PROGRAM MAIN
VAR
END_VAR

FillBox();
Vision();
StartStop();

END_PROGRAM

(* stored: Version 1.1.0.1, ProductVersion 3.1.4024.15
   POU MAIN: Id {b371aa73-8b08-469b-8cce-123a011f0cc4}, SpecialFunc None *)
